FUNCTION_BLOCK LEDdriver
VAR_INPUT
	ledBlink : LEDtype;
	blinkInterval : TIME;
	
	ledChannel : UINT := 1;
END_VAR
VAR_OUTPUT
END_VAR
VAR
	ch1 AT %Q* : BOOL ;
	ch2 AT %Q* : BOOL ;
	ch3 AT %Q* : BOOL ;
	ch4 AT %Q* : BOOL ;
	ch5 AT %Q* : BOOL ;
	ch6 AT %Q* : BOOL ;
	ch7 AT %Q* : BOOL ;
	ch8 AT %Q* : BOOL ;
	
	ch1mode AT %Q* : BOOL;
	ch2mode AT %Q* : BOOL;
	ch3mode AT %Q* : BOOL;
	ch4mode AT %Q* : BOOL;
	ch5mode AT %Q* : BOOL;
	ch6mode AT %Q* : BOOL;
	ch7mode AT %Q* : BOOL;
	ch8mode AT %Q* : BOOL;
	
	tmr1 : TON;
	
	value : BOOL := FALSE;
	currentValue : BOOL := FALSE;
	executed : BOOL := FALSE;
END_VAR

CASE ledChannel OF
	1:
		currentValue := ch1;
	2:
		currentValue := ch2;
	3:
		currentValue := ch3;
	4:
		currentValue := ch4;
	5:
		currentValue := ch5;
	6:
		currentValue := ch6;
	7:
		currentValue := ch7;
	8:
		currentValue := ch8;
END_CASE

CASE ledBlink OF
	LEDtype.OFF:
		value := FALSE;
		executed := FALSE;
	LEDtype.ON:
		value := TRUE;
	LEDtype.BlinkOnce:
		IF currentValue AND tmr1.Q THEN
			value := FALSE;
			tmr1(IN := FALSE);
			executed := TRUE;
		ELSIF NOT executed THEN
			value := TRUE;
			tmr1(IN := TRUE, PT := T#0.5S);
		END_IF
	LEDtype.BlinkContinious:
		IF currentValue AND tmr1.Q THEN
			value := FALSE;
			tmr1(IN := FALSE);
			tmr1(IN := TRUE, PT := blinkInterval);
			executed := TRUE;
		ELSIF NOT currentValue AND tmr1.Q THEN
			value := TRUE;
			tmr1(IN := FALSE);
			tmr1(IN := TRUE, PT := blinkInterval);
		ELSIF NOT executed THEN
			executed := TRUE;
			tmr1(IN := TRUE, PT := T#0.01S);
		ELSE
			tmr1();
		END_IF
	LEDtype.Pulse:
		IF currentValue AND tmr1.Q THEN
			value := FALSE;
			tmr1(IN := FALSE);
			tmr1(IN := TRUE, PT := blinkInterval);
			executed := TRUE;
		ELSIF NOT currentValue AND tmr1.Q THEN
			value := TRUE;
			tmr1(IN := FALSE);
			tmr1(IN := TRUE, PT := T#0.01S);
		ELSIF NOT executed THEN
			executed := TRUE;
			tmr1(IN := TRUE, PT := T#0.01S);
		ELSE
			tmr1();
		END_IF
END_CASE

CASE ledChannel OF
	1:
		ch1mode := TRUE;
		ch1 := value;
	2:
		ch2mode := TRUE;
		ch2 := value;
	3:
		ch3mode := TRUE;
		ch3 := value;
	4:
		ch4mode := TRUE;
		ch4 := value;
	5:
		ch5mode := TRUE;
		ch5 := value;
	6:
		ch6mode := TRUE;
		ch6 := value;
	7:
		ch7mode := TRUE;
		ch7 := value;
	8:
		ch8mode := TRUE;
		ch8 := value;
	9:
		ch1mode := FALSE;
		ch2mode := FALSE;
		ch3mode := FALSE;
		ch4mode := FALSE;
		ch5mode := FALSE;
		ch6mode := FALSE;
		ch7mode := FALSE;
		ch8mode := FALSE;
END_CASE

END_FUNCTION_BLOCK

(* stored: Version 1.1.0.1, ProductVersion 3.1.4022.18
   POU LEDdriver: Id {63d6069d-0186-49e2-85bb-3117e0ee761d}, SpecialFunc None *)
